// TIA Portal V18 export
FUNCTION "Interlocks" : Void   // FC1, SCL
{ S7_Optimized_Access := 'TRUE' }
VERSION : 0.1
// stored: AutoNumber true, IsIECCheckEnabled false, SetENOAutomatically false, UDAEnableTagReadback false
   VAR_INPUT
      capacitive_HLS : Bool;
      temperature : Int;
      emergency_state : Bool;
      FCV_valve_closed : Bool;
      ESD_valve_closed : Bool;
      grounding : Bool;
      Temperature_threshold : Real;
   END_VAR
   VAR_OUTPUT
      temperature_is_ok : Bool;
      interlocks : Bool;
   END_VAR
BEGIN

   //High level,Pendant emergency stop, panel emergency Stop sensors are Normally close

   // Temperature, divided by ten because it the program it shows it 10x
   #temperature_is_ok := #temperature / 10 < #Temperature_threshold;

   //"Interlocks
   IF
       #temperature_is_ok
       AND #emergency_state
       AND #FCV_valve_closed
       AND #ESD_valve_closed
       AND #grounding
   THEN

       #interlocks := 1;
   ELSE
       #interlocks := 0;
   END_IF;
END_FUNCTION
